PROGRAM MAIN
VAR
	numFactorial : ULINT;
	resFactorial : ULINT;
	setBool : BOOL;
END_VAR

IF setBool THEN
	resFactorial := IO.F_factorial(n := numFactorial);
	setBool := FALSE;	
END_IF

END_PROGRAM

(* stored: Version 1.1.0.1, ProductVersion 3.1.4024.12
   POU MAIN: Id {e9a7dbc3-4bf2-4892-888c-7d3496da100e}, SpecialFunc None *)
